Staubli VAL3: calc_score.pgx

program calc_score()
  local num l_nElement
begin

  append(nCompletion)

  for l_nElement = (size(sQueue)-1) to 0 step -1

    if sQueue[l_nElement] == "("
      nCompletion[size(nCompletion)-2] = 5*nCompletion[size(nCompletion)-2] + 1
    endIf
    if sQueue[l_nElement] == "["
      nCompletion[size(nCompletion)-2] = 5*nCompletion[size(nCompletion)-2] + 2
    endIf
    if sQueue[l_nElement] == "{"
      nCompletion[size(nCompletion)-2] = 5*nCompletion[size(nCompletion)-2] + 3
    endIf
    if sQueue[l_nElement] == "<"
      nCompletion[size(nCompletion)-2] = 5*nCompletion[size(nCompletion)-2] + 4
    endIf

  endFor


end
